{attribute 'linkalways'} 
{attribute 'no_explicit_call' := 'This FB is a CLASS and must be accessed using methods or properties'}
{attribute 'enable_dynamic_creation'}
FUNCTION_BLOCK FINAL ADD_INT EXTENDS Node
VAR
	in1 : _INT(0);
	in2 : _INT(0);
	out : _INT(0);
END_VAR

METHOD PUBLIC Clone : I_Node
VAR
	pNode : POINTER TO ADD_INT;
END_VAR
pNode := __NEW(ADD_INT);
Clone := pNode^;
END_METHOD

METHOD FB_init : BOOL
VAR_INPUT
	bInitRetains : BOOL; // if TRUE, the retain variables are initialized (warm start / cold start)
	bInCopyCode : BOOL;  // if TRUE, the instance afterwards gets moved into the copy code (online change)
END_VAR
AddInput('in1',THIS^.in1);
AddInput('in2',THIS^.in2);
AddOutput('out', THIS^.out);
END_METHOD

METHOD PROTECTED OnExecute
VAR
END_VAR
out.Value := in1.Value + in2.Value;
END_METHOD

END_FUNCTION_BLOCK

(* stored: Version 1.1.0.1, ProductVersion 3.1.4024.15
   POU ADD_INT: Id {5c6e1b49-448c-4006-97c0-af63ce645303}, SpecialFunc None
   Folder Constructor: Id {9bb40add-2ec7-4ef3-8661-ad6d30a01d72}
   Method Clone: Id {95b06bd0-7596-4b41-9b58-8d9ac959cb73}
   Method FB_init: Id {f721b957-92e8-4362-9aff-27597882b6ea}
   Method OnExecute: Id {9664ce6b-e5fa-4939-bdb3-b005b3f2b2e4} *)
